RoboDK station: test station.rdk

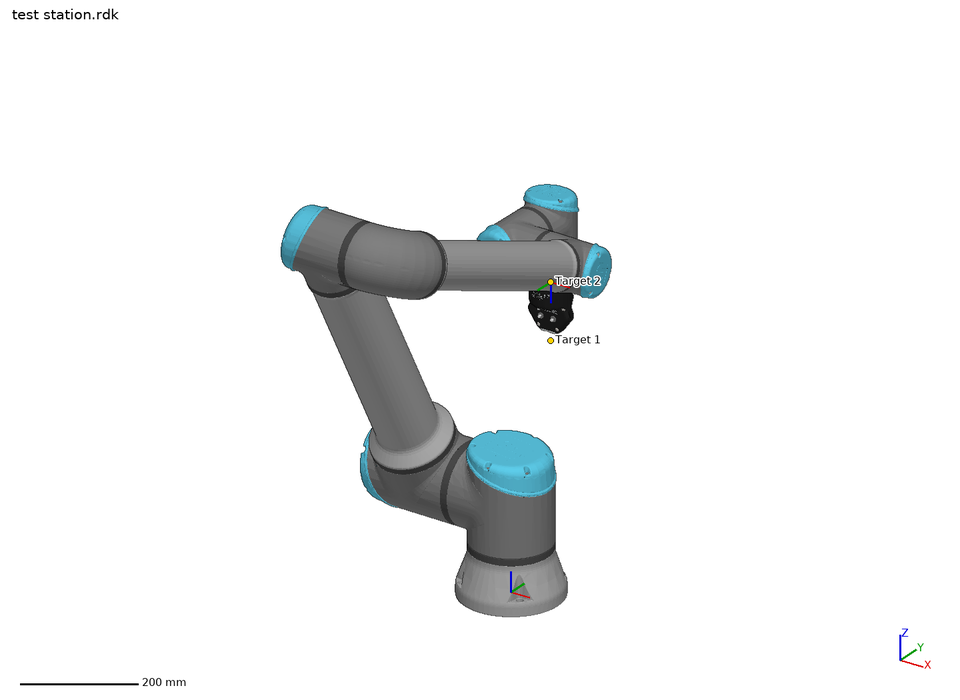
[picture v0: the station drawn from its stored meshes, robots at their saved joint values, targets as dots, program paths as lines]
Station test station (saved by RoboDK 5.6.1). Poses are relative to the parent item; angles as X-Y-Z fixed-axis rotations.
  - frame UR10e Base at (0, 0, 0) mm
    - robot UR10e: 6 axes, payload 10 kg, reach 1300 mm, repeatability 0.05 mm, weight 28.9 kg
        modified DH rows (alpha deg, a mm, theta deg, d mm): 0, 0, 0, 180.7; 90, 0, 180, 0; 0, 612.6, 0, 0; 0, 571.335, 0, 174.15; -90, 0, 0, 119.85; 90, 0, 180, 116.55
        joint limits [-360, -360, -360, -360, -360, -360] to [360, 360, 360, 360, 360, 360]; home [0, -90, -90, 0, 90, 0]; saved at [269.484, -118.233, 140.085, -111.867, 270.077, -0.817]
      - frame RobotiQ 2F-85 Gripper (Mechanism) Base at (0, 0, 0) mm
        - robot RobotiQ 2F-85 Gripper (Mechanism) (model RobotiQ 2F85): 1 axes, payload 5 kg
            joint limits [0] to [85]; home [85]; saved at [85]
    - target Target 1 (joint target) at (-171.04, 361.92, 281.33) mm, rotated rx -179.98 ry 0.08 rz 0.3 deg; joints [269.482, -109.281, 148.481, -129.22, 270.076, -0.818] of UR10e
    - target Target 2 (joint target) at (-171.04, 361.92, 391.33) mm, rotated rx -179.98 ry 0.08 rz 0.3 deg; joints [269.482, -118.24, 140.08, -111.861, 270.075, -0.817] of UR10e
  - Python program Program (listed below)

--- Python program Program ---
import time
import os

from robodk import robolink    # RoboDK API
from robodk import robomath    # Robot toolbox
from robodk.robolink import ITEM_TYPE_ROBOT, ITEM_TYPE_TARGET

RDK = robolink.Robolink()
RDK.setRunMode(6)
from robodk import *      # RoboDK API
from robolink import *    # Robot toolbox

# Get the robot item from the RoboDK station
robot = RDK.Item('UR10e', ITEM_TYPE_ROBOT)

while(1):
    target1 = RDK.Item('Target 1')
    target1 = target1.Joints().list()
    print(target1)

    pause(3)
    ## Getting Current Joint Value
    getJoints = robot.Joints().list()
    print(getJoints)


    ## Moving Robot to Start Position
    if getJoints != target1:
        print("Moving Robot to Target 1")
        try:
            robot.MoveL(target1)
        except:
            pause(5)
        finally:
            robot.MoveL(target1)
    else:
        print("Robot is at Target 1")

    # Gripper Open
    RDK.Disconnect()
    pause(2)
    os.system('python "C:/Users/Syed.bukhari/OneDrive - AddQual/Desktop/Mustafa/Gripper_Scripts/GripperOpen.py"')
    pause(3)
    RDK.Connect()
    RDK.setRunMode(6)

    # Getting Target 2
    target2 = RDK.Item('Target 2')
    target2 = target2.Joints().list()
    print(target2)

    ## Getting Current Joint Value
    getJoints = robot.Joints().list()
    print(getJoints)


    ## Moving Robot to Start Position
    if getJoints != target2:
        print("Moving Robot to Target 2")
        try:
            robot.MoveL(target2)
        except:
            pause(5)
        finally:
            robot.MoveL(target2)

    else:
        print("Robot is at Target 2")

    # Gripper Close
    RDK.Disconnect()
    pause(2)
    os.system('python "C:/Users/Syed.bukhari/OneDrive - AddQual/Desktop/Mustafa/Gripper_Scripts/GripperClose.py"')
    pause(3)
    RDK.Connect()
    RDK.setRunMode(6)
